TEXTLIST TL_FbStateCS
  0 = 'UNDEFINED'
  1 = 'RUN'
  2 = 'STOP'
  3 = 'SAFE'
  4 = 'ERROR'
  5 = 'RESET'
  10 = 'ACTIVE'
  11 = 'DEACTIVE'
   = ''
END_TEXTLIST

(* stored: Version 1.1.0.1, ProductVersion 3.1.4022.12
   TextList TL_FbStateCS: Id {1124f122-601f-4726-8c61-bf6651053380} *)
